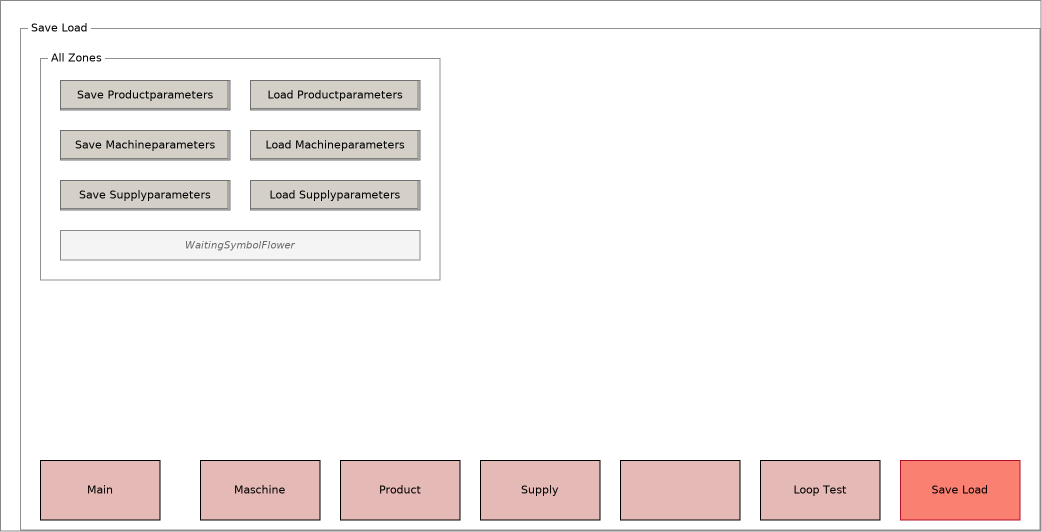
VISUALIZATION Visu_SaveLoad  // 1042x532
    GroupBox (20,20 1020x510), "Save Load"
        Rectangle (20,440 120x60), "Main"
            OnMouseClick: change screen: Visu_Main
        GroupBox (20,30 400x230), "All Zones", input disabled if: stTempSave.stTempCmd.bSaveMparams OR stTempSave.stTempCmd.bSaveSupplyParams OR stTempSave.stTempCmd.bSavePparams OR stTempLoad.stTempCmd.bLoadMparams OR stTempLoad.stTempCmd.bLoadPparams OR stTempLoad.stTempCmd.bLoadSupplyParams
            Button (20,30 170x30), "Save Productparameters"
                toggle stTempSave.stTempCmd.bSavePparams
            Button (210,30 170x30), "Load Productparameters"
                toggle stTempLoad.stTempCmd.bLoadPparams
            Button (20,80 170x30), "Save Machineparameters"
                toggle stTempSave.stTempCmd.bSaveMparams
            Button (210,80 170x30), "Load Machineparameters"
                toggle stTempLoad.stTempCmd.bLoadMparams
            Button (20,130 170x30), "Save Supplyparameters"
                toggle stTempSave.stTempCmd.bSaveSupplyParams
            Button (210,130 170x30), "Load Supplyparameters"
                toggle stTempLoad.stTempCmd.bLoadSupplyParams
            WaitingSymbolFlower (20,180 360x30), invisible if: NOT(stTempSave.stTempCmd.bSaveMparams OR stTempSave.stTempCmd.bSaveSupplyParams OR stTempSave.stTempCmd.bSavePparams OR stTempLoad.stTempCmd.bLoadMparams OR stTempLoad.stTempCmd.bLoadPparams OR stTempLoad.stTempCmd.bLoadSupplyParams)
        Rectangle (880,440 120x60), "Save Load"
            OnMouseClick: change screen: Visu_SaveLoad
        Rectangle (320,440 120x60), "Product"
            OnMouseClick: change screen: Visu_PParam
        Rectangle (180,440 120x60), "Maschine"
            OnMouseClick: change screen: Visu_MParam
        Rectangle (460,440 120x60), "Supply"
            OnMouseClick: change screen: Visu_Supply
        Rectangle (600,440 120x60)
        Rectangle (740,440 120x60), "Loop Test"
            OnMouseClick: change screen: Visu_LoopTest
END_VISUALIZATION

(* stored: Version 1.1.0.1, ProductVersion 3.1.4024.12
   Visu Visu_SaveLoad: Id {c77f5c7b-a6d0-4ed3-aebb-22dca497e3f1} *)
